FUNCTION_BLOCK FB_Event EXTENDS FB_ListString IMPLEMENTS I_Event
VAR_INPUT
	bIngoreHold:			BOOL:= TRUE;
	bIngorePause:			BOOL:= TRUE;
END_VAR
VAR_OUTPUT
END_VAR
VAR
	iParent:			I_Component;
	iLogger:			I_Logger;
	stError:			ST_Event;
	stWarning:			ST_Event;
	stInformation:		ST_Event;
	stDebug:			ST_Event;
END_VAR

SUPER^();

METHOD FB_init : BOOL
VAR_INPUT
	bInitRetains : BOOL; // if TRUE, the retain variables are initialized (warm start / cold start)
	bInCopyCode : BOOL;  // if TRUE, the instance afterwards gets moved into the copy code (online change)
	iParent:			I_Component;
END_VAR
THIS^.iParent:= iParent;
END_METHOD

METHOD INTERNAL M_Arguments : STRING(255)
VAR_INPUT
END_VAR
VAR
	nIndex:			INT;
END_VAR
WHILE nIndex < nLength DO
	M_Arguments:= Concat(Concat(M_Arguments, pList[nIndex]), '$N');
	nIndex:= nIndex + 1;
END_WHILE
END_METHOD

METHOD PUBLIC M_Debug : BOOL
VAR_INPUT
	Message:				STRING(255);
END_VAR
IF stDebug.Message <> Message THEN
	stDebug.New:= TRUE;
ELSE
	stDebug.New:= FALSE;
END_IF

stDebug.Source:= iParent;
stDebug.Instance:= iParent.P_Info.P_Instance;
stDebug.Class:= iParent.P_Info.P_Class;
stDebug.EventType:= E_Event.Debug;
stDebug.Timestamp:= F_GetSystemTime();
stDebug.ID:= 0;
stDebug.Message:= Message;
stDebug.Arguments:= M_Arguments();
stDebug.Active:= TRUE;

IF iLogger <> 0 THEN
	iLogger.M_Log(stDebug);
END_IF

M_Clear();
END_METHOD

METHOD PUBLIC M_Error : BOOL
VAR_INPUT
	Message:				STRING(255);
	ID:						UDINT;
	Behaviour:				E_Behaviour;
END_VAR
IF stError.Message <> Message THEN
	stError.Source:= iParent;
	stError.Instance:= iParent.P_Info.P_Instance;
	stError.Class:= iParent.P_Info.P_Class;
	stError.EventType:= E_Event.Error;
	stError.Timestamp:= F_GetSystemTime();
	stError.ID:= ID;
	stError.Message:= Message;
	stError.Arguments:= M_Arguments();
	stError.New:= TRUE;
	stError.Active:= TRUE;


	IF Behaviour >= E_Behaviour.Abort THEN
		iParent.M_Request(E_Request.Abort);
	ELSIF Behaviour >= E_Behaviour.Stop THEN
		iParent.M_Request(E_Request.Stop);
	ELSIF Behaviour >= E_Behaviour.Complete THEN	
		iParent.M_Request(E_Request.Complete);
	ELSIF Behaviour >= E_Behaviour.Hold THEN
		iParent.M_Request(E_Request.Hold);
	ELSIF Behaviour >= E_Behaviour.Pause THEN
		iParent.M_Request(E_Request.Pause);
	END_IF
	
	IF iLogger <> 0 THEN
		iLogger.M_Log(stError);
	END_IF
END_IF

M_Clear();
END_METHOD

METHOD PUBLIC M_Information : BOOL
VAR_INPUT
	Message:				STRING(255);
	ID:						UDINT;
END_VAR
IF stInformation.Message <> Message THEN
	stInformation.New:= TRUE;
ELSE
	stInformation.New:= FALSE;
END_IF

stInformation.Source:= iParent;
stInformation.Instance:= iParent.P_Info.P_Instance;
stInformation.Class:= iParent.P_Info.P_Class;
stInformation.EventType:= E_Event.Information;
stInformation.Timestamp:= F_GetSystemTime();
stInformation.ID:= ID;
stInformation.Message:= Message;
stInformation.Arguments:= M_Arguments();
stInformation.Active:= TRUE;

IF iLogger <> 0 THEN
	iLogger.M_Log(stInformation);
END_IF

M_Clear();
END_METHOD

METHOD PUBLIC M_Reset
VAR_INPUT
END_VAR
Memset(ADR(stError), 0, SIZEOF(stError));
Memset(ADR(stWarning), 0, SIZEOF(stWarning));
Memset(ADR(stInformation), 0, SIZEOF(stInformation));
Memset(ADR(stDebug), 0, SIZEOF(stDebug));
END_METHOD

METHOD PUBLIC M_Warning : BOOL
VAR_INPUT
	Message:				STRING(255);
	ID:						UDINT;
END_VAR
IF stWarning.Message <> Message THEN
	stWarning.New:= TRUE;
ELSE
	stWarning.New:= FALSE;
END_IF

stWarning.Source:= iParent;
stWarning.Instance:= iParent.P_Info.P_Instance;
stWarning.Class:= iParent.P_Info.P_Class;
stWarning.EventType:= E_Event.Warning;
stWarning.Timestamp:= F_GetSystemTime();
stWarning.ID:= ID;
stWarning.Message:= Message;
stWarning.Arguments:= M_Arguments();
stWarning.Active:= TRUE;

IF iLogger <> 0 THEN
	iLogger.M_Log(stWarning);
END_IF

M_Clear();
END_METHOD

PROPERTY PUBLIC P_Logger : I_Logger
GET
P_Logger:= iLogger;
END_GET
SET
iLogger:= P_Logger;
END_SET
END_PROPERTY

END_FUNCTION_BLOCK

(* stored: Version 1.1.0.1
   POU FB_Event: Id {59616103-7f2e-4b6f-81bd-583969a36d28}, SpecialFunc None
   Method FB_init: Id {be23ffcc-529d-4010-ace3-b17baed191a5}
   Method M_Arguments: Id {70779266-7b36-4bce-9e6f-049e951fd75a}
   Method M_Debug: Id {0a2b992b-2a4a-0251-0210-713b326debf6}
   Method M_Error: Id {55348828-4763-4c06-9dd1-090fa29a8379}
   Method M_Information: Id {d9a244f2-1d6f-434f-aab4-cad6aacbb94f}
   Method M_Reset: Id {31d9e5bb-2957-4381-81b6-d0453bdac8d3}
   Method M_Warning: Id {d443b8bb-774e-487e-80a2-79cf66a0376c}
   Property P_Logger: Id {642d0edf-ded0-4248-be29-8384d3180124}
   Get Get: Id {99e41819-eb78-4b29-b3e9-6728532b14b1}
   Set Set: Id {be31597a-6e88-476b-aec8-980317d6bc1a} *)
